// Mitsubishi GX Works2 project: plc_group6_PART2   PLC: FX3G

// global labels: Global1
VAR_GLOBAL
  sen_door AT X000 : BOOL;
  system_on AT M0 : BOOL;
  timer_10_min AT TC1 : BOOL;
END_VAR
VAR_GLOBAL CONSTANT
  min_10 : INT := 6000;
END_VAR
VAR_GLOBAL
  massage_start AT Y003 : BOOL;
  timer_10_min_ts1 AT TS1 : BOOL;
  system_on_switch AT X001 : BOOL;
  timer_20_min AT TC2 : BOOL;
END_VAR
VAR_GLOBAL CONSTANT
  min_20 : INT := 12000;
END_VAR
VAR_GLOBAL
  timer_20_min_ts2 AT TS2 : BOOL;
  timer_30_min_ts3 AT TS3 : BOOL;
  massage_faster AT Y004 : BOOL;
  timer_30_min AT TC3 : BOOL;
END_VAR
VAR_GLOBAL CONSTANT
  min_30 : INT := 18000;
END_VAR

// task Task_01 (event TRUE, interval 0, priority 31): POU_01

PROGRAM POU_01
(* structured ladder/FBD written out as ST: instructions are called as NAME(EN, inputs, outputs); _pN, _eN, _tN stand for wires *)
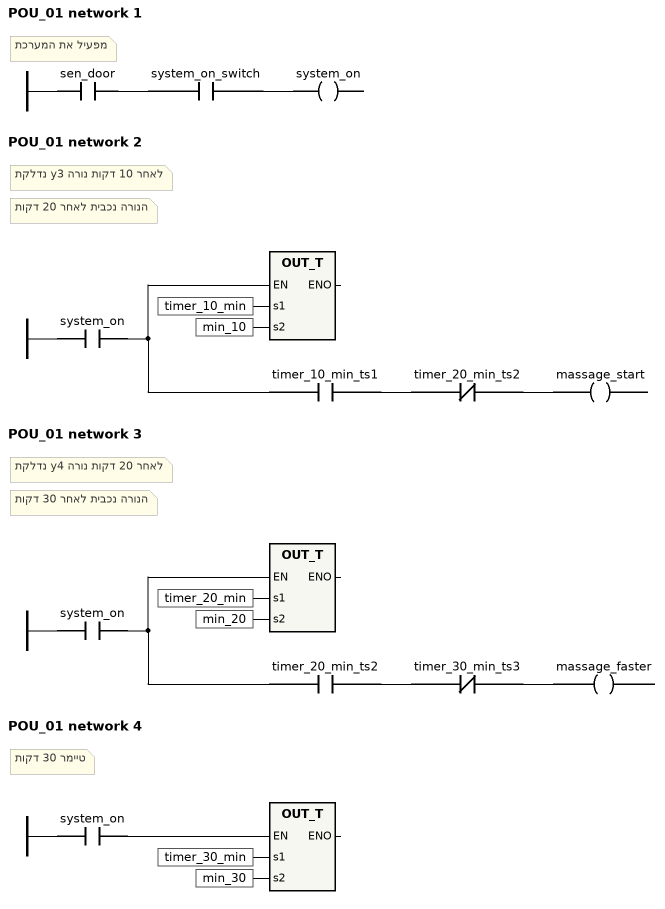
(* network 1 *)
(* מפעיל את המערכת *)
system_on := sen_door AND system_on_switch;
(* network 2 *)
(* לאחר 10 דקות נורה y3 נדלקת *)
(* הנורה נכבית לאחר 20 דקות *)
OUT_T(system_on, timer_10_min, min_10);
massage_start := system_on AND timer_10_min_ts1 AND NOT timer_20_min_ts2;
(* network 3 *)
(* לאחר 20 דקות נורה y4 נדלקת *)
(* הנורה נכבית לאחר 30 דקות *)
OUT_T(system_on, timer_20_min, min_20);
massage_faster := system_on AND timer_20_min_ts2 AND NOT timer_30_min_ts3;
(* network 4 *)
(* טיימר 30 דקות *)
OUT_T(system_on, timer_30_min, min_30);
END_PROGRAM
